PROGRAM EM01_BoxInfeed
VAR
//----Motor-----
	// Box Buffer Roller Conveyor 1	
	FB_BoxBufferRollerConv_1			: MotorManagement;
	stBoxBufferRollerConv_1				: stMotor;
	BoxBufferRollerConv_1_ErrorID		: UINT;
	BoxBufferRollerConv_1_Error			: BOOL;
	bFL_BoxBufferRollerConv_1_Forward	: BOOL;
	// Box Buffer Roller Conveyor 2	
	FB_BoxBufferRollerConv_2			: MotorManagement;
	stBoxBufferRollerConv_2				: stMotor;
	BoxBufferRollerConv_2_ErrorID		: UINT;
	BoxBufferRollerConv_2_Error			: BOOL;
	bFL_BoxBufferRollerConv_2_Forward	: BOOL;
	// Box Stop & Go Belt Conveyor
	FB_BoxStopEndGoBeltConv				: MotorManagement;
	stBoxStopEndGoBeltConv				: stMotor;
	BoxStopEndGoBeltConv_ErrorID		: UINT;
	BoxStopEndGoBeltConv_Error			: BOOL;
	bFL_BoxStopEndGoBeltConv_Forward	: BOOL;
	// Box Picking Roller Conveyor
	FB_BoxPickingRollerConv				: MotorManagement;
	stBoxPickingRollerConv				: stMotor;
	BoxPickingRollerConv_ErrorID		: UINT;
	BoxPickingRollerConv_Error			: BOOL;
	bFL_BoxPickingRollerConv_Forward	: BOOL;
END_VAR

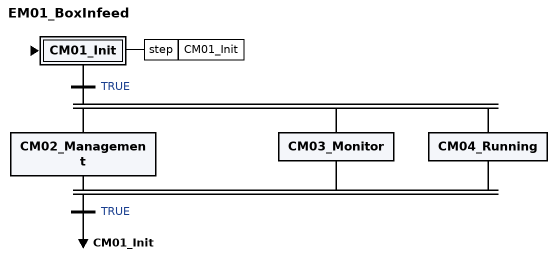
INITIAL_STEP CM01_Init:
    CM01_Init(N);  // step action
END_STEP
TRANSITION FROM CM01_Init TO (CM02_Management, CM03_Monitor, CM04_Running)
    := TRUE;
END_TRANSITION
STEP CM02_Management:
END_STEP
STEP CM03_Monitor:
END_STEP
STEP CM04_Running:
END_STEP
TRANSITION FROM (CM02_Management, CM03_Monitor, CM04_Running) TO CM01_Init
    := TRUE;
END_TRANSITION

ACTION CM01_Init:

END_ACTION

ACTION CM02_Management:
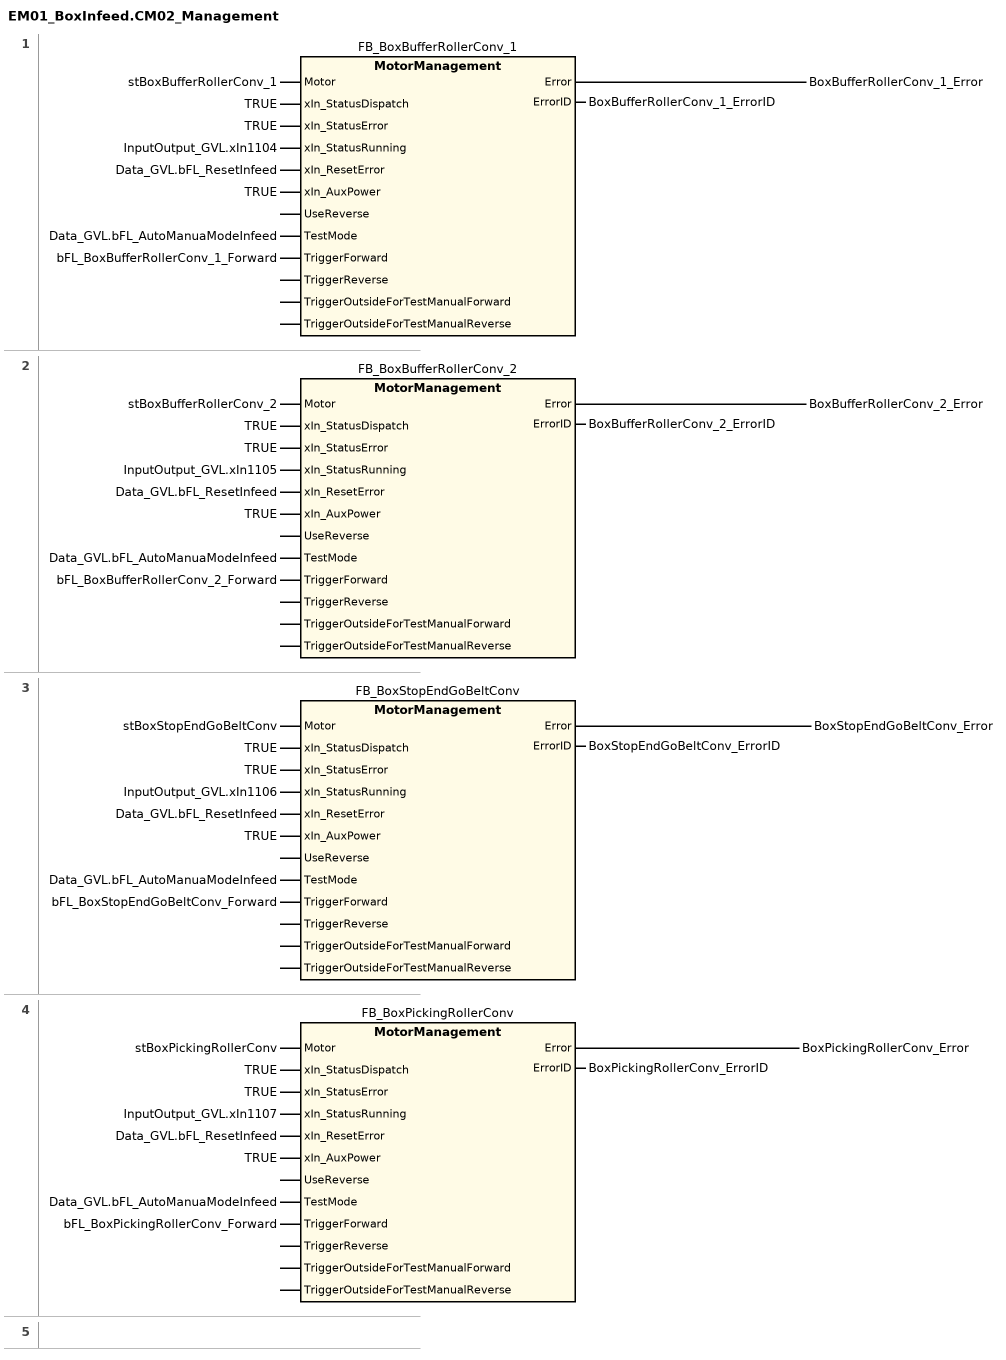
// NETWORK 1
FB_BoxBufferRollerConv_1(
    Motor := stBoxBufferRollerConv_1,
    xIn_StatusDispatch := TRUE,
    xIn_StatusError := TRUE,
    xIn_StatusRunning := InputOutput_GVL.xIn1104,
    xIn_ResetError := Data_GVL.bFL_ResetInfeed,
    xIn_AuxPower := TRUE,
    TestMode := Data_GVL.bFL_AutoManuaModeInfeed,
    TriggerForward := bFL_BoxBufferRollerConv_1_Forward,
    ErrorID => BoxBufferRollerConv_1_ErrorID); // MotorManagement
BoxBufferRollerConv_1_Error := FB_BoxBufferRollerConv_1.Error;

// NETWORK 2
FB_BoxBufferRollerConv_2(
    Motor := stBoxBufferRollerConv_2,
    xIn_StatusDispatch := TRUE,
    xIn_StatusError := TRUE,
    xIn_StatusRunning := InputOutput_GVL.xIn1105,
    xIn_ResetError := Data_GVL.bFL_ResetInfeed,
    xIn_AuxPower := TRUE,
    TestMode := Data_GVL.bFL_AutoManuaModeInfeed,
    TriggerForward := bFL_BoxBufferRollerConv_2_Forward,
    ErrorID => BoxBufferRollerConv_2_ErrorID); // MotorManagement
BoxBufferRollerConv_2_Error := FB_BoxBufferRollerConv_2.Error;

// NETWORK 3
FB_BoxStopEndGoBeltConv(
    Motor := stBoxStopEndGoBeltConv,
    xIn_StatusDispatch := TRUE,
    xIn_StatusError := TRUE,
    xIn_StatusRunning := InputOutput_GVL.xIn1106,
    xIn_ResetError := Data_GVL.bFL_ResetInfeed,
    xIn_AuxPower := TRUE,
    TestMode := Data_GVL.bFL_AutoManuaModeInfeed,
    TriggerForward := bFL_BoxStopEndGoBeltConv_Forward,
    ErrorID => BoxStopEndGoBeltConv_ErrorID); // MotorManagement
BoxStopEndGoBeltConv_Error := FB_BoxStopEndGoBeltConv.Error;

// NETWORK 4
FB_BoxPickingRollerConv(
    Motor := stBoxPickingRollerConv,
    xIn_StatusDispatch := TRUE,
    xIn_StatusError := TRUE,
    xIn_StatusRunning := InputOutput_GVL.xIn1107,
    xIn_ResetError := Data_GVL.bFL_ResetInfeed,
    xIn_AuxPower := TRUE,
    TestMode := Data_GVL.bFL_AutoManuaModeInfeed,
    TriggerForward := bFL_BoxPickingRollerConv_Forward,
    ErrorID => BoxPickingRollerConv_ErrorID); // MotorManagement
BoxPickingRollerConv_Error := FB_BoxPickingRollerConv.Error;

// NETWORK 5
END_ACTION

ACTION CM03_Monitor:
// NETWORK 1
END_ACTION

ACTION CM04_Running:
// NETWORK 1
END_ACTION

END_PROGRAM

(* stored: Version 1.1.0.1, ProductVersion 3.1.4024.9
   POU EM01_BoxInfeed: Id {f969e190-b0d9-4bd0-abef-d434d6bb78f5}, SpecialFunc None
   Action CM01_Init: Id {c1577cd7-8c01-4930-bc0f-171842f749d0}
   Action CM02_Management: Id {04c90148-ee95-46c4-a456-920c69769461}
   Action CM03_Monitor: Id {1562048c-a3dc-491e-a7d5-5c4cdec2add6}
   Action CM04_Running: Id {84dcb06f-9cea-4fe6-bea6-ebcd01c6f315} *)
